FUNCTION_BLOCK SLOT_SIMPLE_ITERATOR (* Iterator *)
  (* Standard: 61499-2 *)
  (* Version 1.0, 27-05-12, GASR, Universidade do Estado de Santa Catarina *)
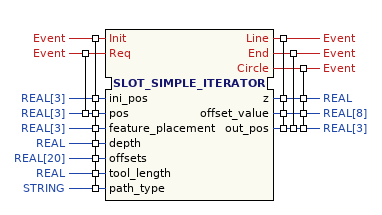
  EVENT_INPUT
    Init WITH ini_pos, pos, feature_placement, depth, offsets, tool_length, path_type;
    Req WITH pos;
  END_EVENT
  EVENT_OUTPUT
    Line WITH z, offset_value, out_pos;
    End WITH out_pos;
    Circle WITH z, offset_value, out_pos;
  END_EVENT
  VAR_INPUT
    ini_pos : ARRAY [0..2] OF REAL;
    pos : ARRAY [0..2] OF REAL;
    feature_placement : ARRAY [0..2] OF REAL;
    depth : REAL;
    offsets : ARRAY [0..19] OF REAL;
    tool_length : REAL;
    path_type : STRING;
  END_VAR
  VAR_OUTPUT
    z : REAL;
    offset_value : ARRAY [0..7] OF REAL;
    out_pos : ARRAY [0..2] OF REAL;
  END_VAR
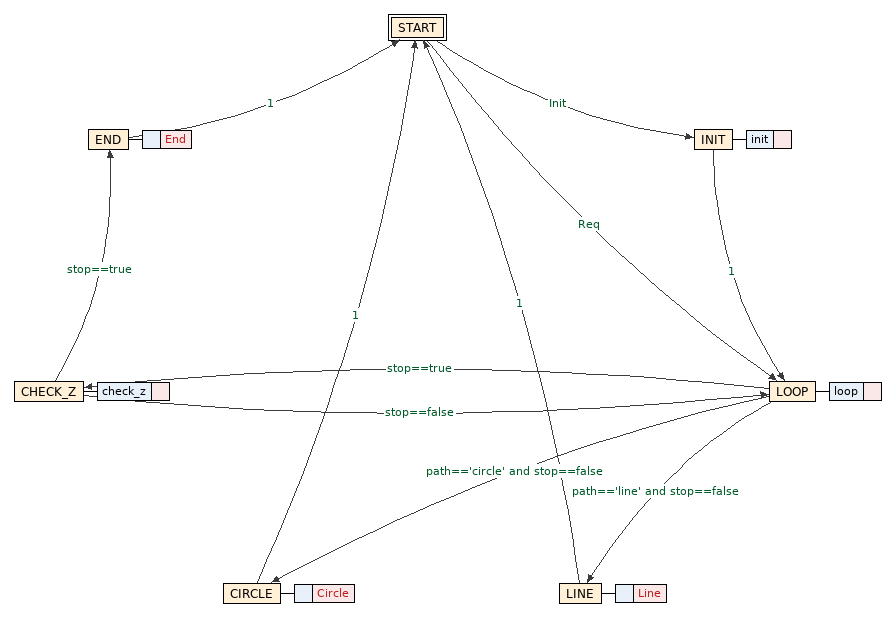
  EC_STATES
    START;
    INIT : init;
    LOOP : loop;
    LINE : -> Line;
    CIRCLE : -> Circle;
    CHECK_Z : check_z;
    END : -> End;
  END_STATES
  EC_TRANSITIONS
    START TO INIT := Init;
    START TO LOOP := Req;
    INIT TO LOOP := 1;
    LOOP TO LINE := path=='line' and stop==false;
    LOOP TO CIRCLE := path=='circle' and stop==false;
    LOOP TO CHECK_Z := stop==true;
    CHECK_Z TO END := stop==true;
    CHECK_Z TO LOOP := stop==false;
    LINE TO START := 1;
    CIRCLE TO START := 1;
    END TO START := 1;
  END_TRANSITIONS
  ALGORITHM init IN Lua:
stop = false
path_iteration = 0
pos[1] = ini_pos[1]
pos[2] = ini_pos[2]
pos[3] = ini_pos[3]
for k, v in ipairs( offsets ) do
    if( type( v ) == 'number' ) then
        offsets[ k ] = nil
    end
end
z = pos[3]
  END_ALGORITHM
  ALGORITHM loop IN Lua:
if( path_iteration >= #offsets  ) then
	stop = true
    out_pos[i] = pos[i]
else
	path_iteration = path_iteration + 1
	for i = 1, #offsets[ path_iteration ] do
		out_pos[i] = pos[i]
		offset_value[i] = offsets[ path_iteration ][i]
	end
	offset_value[3] = z
	print( 'offset size', #offset_value, 'pos', out_pos[1], out_pos[2], out_pos[3] )
	if(( (offset_value[1] - pos[1]) == 0 ) and ( (offset_value[2] - pos[2]) == 0 ) and ( (offset_value[3] - pos[3]) == 0 )) then
        path_iteration = path_iteration + 1
        for i = 1, #offsets[ path_iteration ] do
            offset_value[i] = offsets[ path_iteration ][i]
        end
        offset_value[3] = z
    end
	if( path_type == 'LINEAR_PATH' ) or ((( path_type == 'COMPLETE_CIRCULAR_PATH' ) or ( path_type == 'PARTIAL_CIRCULAR_PATH' )) and ( #offsets[ path_iteration ] == 3 )) then
		path = 'line'
	elseif(( path_type == 'COMPLETE_CIRCULAR_PATH' ) or ( path_type == 'PARTIAL_CIRCULAR_PATH' )) and ( #offsets[ path_iteration ] == 8 ) then
        path = 'circle'
    end
    print( 'path', path, #offset_value, #offsets[ path_iteration ], offset_value[5], path_iteration, '\n' )
end
  END_ALGORITHM
  ALGORITHM check_z IN Lua:
current_z = pos[3]
print( 'iterator', current_z, depth, feature_placement[3], 'pos', pos[1], pos[2], pos[3], depth )
if not( current_z > (depth + feature_placement[3]) ) then
	stop = true
    for i = 1, 3 do
        out_pos[i] = pos[i]
    end
elseif( z == 0 ) then
    stop = false
    for i = 1, 3 do
        out_pos[i] = pos[i]
    end
else
	stop = false
	if( tool_length >= math.abs(depth - current_z) ) then
		z = (current_z + tool_length) + feature_placement[3]
	else
		z = (current_z + (depth - current_z)) + feature_placement[3]
	end
	print( 'new_depth', z )
	path_iteration = 0
end
  END_ALGORITHM
END_FUNCTION_BLOCK
(* other elements stored in the file *)
(* VarDeclaration Name=path_iteration Type=REAL InitialValue=0 *)
(* VarDeclaration Name=stop Type=BOOL InitialValue=false *)
(* VarDeclaration Name=path Type=STRING *)
